TYPE ArduinoLightConfig EXTENDS DeviceConfiguration :
STRUCT
	SerialCommunication : SerialCommunication;
END_STRUCT
END_TYPE

(* stored: Version 1.1.0.1, ProductVersion 3.1.4024.12
   DUT ArduinoLightConfig: Id {f7bed299-4697-44f7-b3fd-e3ac8cdc8282} *)
